{attribute 'GeneratedUsingTerminal: EM7004-0000-9995'}
{attribute addProperty BoxType "EM7004-0000-9995"}
{attribute addProperty Id "StatusAT %I*UINT2ValueAT %I*UINT2LatchAT %I*UINT2"}
{attribute addProperty CRC "776905235"}
{attribute addProperty Size "6"}
TYPE Encoder_Channel_2E4EA213 EXTENDS InputBase_8311D824 :
STRUCT
	{attribute addProperty Name "Status"}
	Status AT %I* : UINT;
	{attribute addProperty Name "Value"}
	Value AT %I* : UINT;
	{attribute addProperty Name "Latch"}
	Latch AT %I* : UINT;
END_STRUCT
END_TYPE

(* stored: Version 1.2.0.0, ProductVersion 3.1.4024.9
   DUT Encoder_Channel_2E4EA213: Id {ef62d1df-e04e-41a6-ad2c-927fb53a1cbd} *)
